screen "输入显示" 800x480
   Rectangle "矩形_2" at 16,42 size 105x25
      Appearance <- "工作台放松压检"
   Rectangle "矩形_1" at 16,14 size 105x25
      Appearance <- "工作台夹紧压检"
   Button "按钮_1" at 28,424 size 67x56; TextOn '滑块角度'; TextOff '滑块角度'
      on Click: ActivateScreen("滑块角度", 0)
   Button "按钮_2" at 96,424 size 67x56; TextOn '设备状态'; TextOff '设备状态'
      on Click: ActivateScreen("设备状态", 0)
   Button "按钮_3" at 163,424 size 71x55; TextOn '工作台操作'; TextOff '工作台操作'
      on Click: ActivateScreen("工作台操作", 0)
   Button "按钮_4" at 235,424 size 69x56; TextOn '气垫操作'; TextOff '气垫操作'
      on Click: ActivateScreen("气垫操作", 0)
   Button "按钮_5" at 304,423 size 66x57; TextOn '故障显示'; TextOff '故障显示'
      on Click: ActivateScreen("故障显示", 0)
   Button "按钮_6" at 371,423 size 73x57; TextOn '输出显示'; TextOff '输出显示'
      on Click: ActivateScreen("输出显示", 0)
   Button "按钮_7" at 445,422 size 66x58; TextOn '输入显示'; TextOff '输入显示'
      on Click: ActivateScreen("输入显示", 0)
   Button "按钮_8" at 514,423 size 68x56; TextOn '滑块调整'; TextOff '滑块调整'
      on Click: ActivateScreen("滑块调整", 0)
   Button "按钮_9" at 592,422 size 65x58; TextOn '报警信息'; TextOff '报警信息'
      on Click: ActivateScreen("报警信息", 0)
   TextField "文本域_1" at 18,20 size 103x17; Text '工作台夹紧压力'
   TextField "文本域_2" at 18,46 size 103x17; Text '工作台放松压力'
   Rectangle "矩形_3" at 16,98 size 105x25
      Appearance <- "平衡缸气压检测"
   Rectangle "矩形_4" at 16,70 size 105x25
      Appearance <- "故障复位"
   Rectangle "矩形_5" at 16,154 size 105x25
      Appearance <- "滑块调整选择"
   Rectangle "矩形_6" at 16,126 size 105x25
      Appearance <- "主电机启动接触器接通"
   Rectangle "矩形_7" at 16,210 size 105x25
      Appearance <- "气垫调整"
   Rectangle "矩形_8" at 16,182 size 105x25
      Appearance <- "行程"
   Rectangle "矩形_9" at 16,266 size 105x25
      Appearance <- "滑块向上"
   Rectangle "矩形_10" at 16,238 size 105x25
      Appearance <- "模具更换"
   TextField "文本域_11" at 36,76 size 61x17; Text '故障复位'
   TextField "文本域_3" at 19,104 size 103x17; Text '平衡缸气压检测'
   TextField "文本域_4" at 15,133 size 105x13; Text '主电机启动接触器接通'
   TextField "文本域_5" at 23,160 size 89x17; Text '滑块调整选择'
   TextField "文本域_6" at 48,188 size 33x17; Text '行程'
   TextField "文本域_7" at 33,215 size 61x17; Text '气垫调整'
   TextField "文本域_8" at 32,243 size 61x17; Text '模具更换'
   TextField "文本域_9" at 32,271 size 61x17; Text '滑块向上'
   Rectangle "矩形_11" at 16,294 size 105x25
      Appearance <- "滑块向下"
   Rectangle "矩形_12" at 16,322 size 105x25
      Appearance <- "停上死点"
   Rectangle "矩形_13" at 16,350 size 105x25
      Appearance <- "滑块调整过扭矩"
   TextField "文本域_10" at 32,300 size 61x17; Text '滑块向下'
   TextField "文本域_12" at 32,327 size 61x17; Text '停上死点'
   TextField "文本域_13" at 17,356 size 103x17; Text '滑块调整过扭矩'
   Rectangle "矩形_14" at 16,377 size 105x25
      Appearance <- "液压保护卸荷"
   TextField "文本域_14" at 23,383 size 89x17; Text '液压保护卸荷'
   Rectangle "矩形_15" at 132,42 size 105x25
      Appearance <- "爬梯开关"
   Rectangle "矩形_16" at 132,14 size 105x25
      Appearance <- "液压保护压力检测"
   Rectangle "矩形_17" at 132,98 size 105x25
      Appearance <- "润滑启动按钮"
   Rectangle "矩形_18" at 132,70 size 105x25
      Appearance <- "润滑停止按钮"
   Rectangle "矩形_19" at 132,154 size 105x25
      Appearance <- "平衡缸手动润滑按钮"
   Rectangle "矩形_20" at 132,126 size 105x25
      Appearance <- "气垫手动润滑按钮"
   Rectangle "矩形_21" at 132,210 size 105x25
      Appearance <- "液压保护复位2"
   Rectangle "矩形_22" at 132,182 size 105x25
      Appearance <- "液压保护复位1"
   Rectangle "矩形_23" at 132,266 size 105x25
      Appearance <- "模具松开按钮"
   Rectangle "矩形_24" at 132,238 size 105x25
      Appearance <- "模具夹紧按钮"
   Rectangle "矩形_25" at 132,294 size 105x25
      Appearance <- "模具更换转换"
   Rectangle "矩形_26" at 132,322 size 105x25
      Appearance <- "工作台夹紧"
   Rectangle "矩形_27" at 132,350 size 105x25
      Appearance <- "工作台松开"
   Rectangle "矩形_28" at 132,377 size 105x25
      Appearance <- "微调启动按钮"
   Rectangle "矩形_29" at 248,42 size 105x25
      Appearance <- "微调反转"
   Rectangle "矩形_30" at 248,14 size 105x25
      Appearance <- "微调正转"
   Rectangle "矩形_31" at 248,98 size 105x25
      Appearance <- "主电机启动1"
   Rectangle "矩形_32" at 248,70 size 105x25
      Appearance <- "主电机停止"
   Rectangle "矩形_33" at 248,154 size 105x25
      Appearance <- "主电机启动2"
   Rectangle "矩形_34" at 248,126 size 105x25
      Appearance <- "微调选择(1)"
   Rectangle "矩形_35" at 248,210 size 105x25
      Appearance <- "寸动闭点1"
   Rectangle "矩形_36" at 248,182 size 105x25
      Appearance <- "寸动开点1"
   Rectangle "矩形_37" at 248,266 size 105x25
      Appearance <- "寸动闭点2"
   Rectangle "矩形_38" at 248,238 size 105x25
      Appearance <- "寸动开点2"
   Rectangle "矩形_39" at 248,294 size 105x25
      Appearance <- "寸动选择"
   Rectangle "矩形_40" at 248,322 size 105x25
      Appearance <- "单次选择"
   Rectangle "矩形_41" at 248,350 size 105x25
      Appearance <- "连续选择"
   Rectangle "矩形_42" at 248,377 size 105x25
      Appearance <- "急停闭点"
   Rectangle "矩形_43" at 364,42 size 105x25
      Appearance <- "急停开点2"
   Rectangle "矩形_44" at 364,14 size 105x25
      Appearance <- "急停开点1"
   Rectangle "矩形_45" at 364,98 size 105x25
      Appearance <- "润滑油位低"
   Rectangle "矩形_46" at 364,70 size 105x25
      Appearance <- "润滑油位高"
   Rectangle "矩形_47" at 364,154 size 105x25
      Appearance <- "润滑低压2"
   Rectangle "矩形_48" at 364,126 size 105x25
      Appearance <- "润滑低压1"
   Rectangle "矩形_49" at 364,210 size 105x25
      Appearance <- "润滑高压"
   Rectangle "矩形_50" at 364,182 size 105x25
      Appearance <- "润滑低压3"
   Rectangle "矩形_51" at 364,266 size 105x25
      Appearance <- "滤油器堵塞2"
   Rectangle "矩形_52" at 364,238 size 105x25
      Appearance <- "滤油器堵塞1"
   Rectangle "矩形_53" at 364,294 size 105x25
      Appearance <- "滤油器堵塞3"
   Rectangle "矩形_54" at 364,322 size 105x25
      Appearance <- "工作台落到位前(1)"
   Rectangle "矩形_55" at 364,350 size 105x25
      Appearance <- "工作台落到位后(1)"
   Rectangle "矩形_56" at 364,377 size 105x25
      Appearance <- "气垫落到位"
   TextField "文本域_15" at 131,19 size 109x16; Text '液压保护压力检测'
   TextField "文本域_16" at 146,47 size 61x17; Text '爬梯开关'
   TextField "文本域_17" at 137,75 size 89x17; Text '润滑停止按钮'
   TextField "文本域_18" at 138,104 size 89x17; Text '润滑启动按钮'
   TextField "文本域_19" at 131,130 size 109x16; Text '气垫手动润滑按钮'
   TextField "文本域_20" at 128,159 size 113x15; Text '平衡缸手动润滑按钮'
   TextField "文本域_21" at 138,187 size 97x17; Text '液压保护复位1'
   TextField "文本域_22" at 137,215 size 97x17; Text '液压保护复位2'
   TextField "文本域_23" at 139,244 size 89x17; Text '模具夹紧按钮'
   TextField "文本域_24" at 139,272 size 89x17; Text '模具松开按钮'
   TextField "文本域_25" at 139,299 size 89x17; Text '模具更换转换'
   TextField "文本域_26" at 142,327 size 75x17; Text '工作台夹紧'
   TextField "文本域_27" at 141,354 size 75x17; Text '工作台松开'
   TextField "文本域_28" at 139,382 size 89x17; Text '微调启动按钮'
   TextField "文本域_29" at 267,20 size 61x17; Text '微调正转'
   TextField "文本域_30" at 267,47 size 61x17; Text '微调反转'
   TextField "文本域_31" at 261,75 size 75x17; Text '主电机停止'
   TextField "文本域_32" at 260,104 size 83x17; Text '主电机启动1'
   TextField "文本域_33" at 260,131 size 85x17; Text '微调选择(1)'
   TextField "文本域_34" at 262,159 size 83x17; Text '主电机启动2'
   TextField "文本域_35" at 267,188 size 69x17; Text '寸动开点1'
   TextField "文本域_36" at 267,216 size 69x17; Text '寸动闭点1'
   TextField "文本域_37" at 266,243 size 69x17; Text '寸动开点2'
   TextField "文本域_38" at 265,271 size 69x17; Text '寸动闭点2'
   TextField "文本域_39" at 268,299 size 61x17; Text '寸动选择'
   TextField "文本域_40" at 270,329 size 61x17; Text '单次选择'
   TextField "文本域_41" at 270,354 size 61x17; Text '连续选择'
   TextField "文本域_42" at 269,382 size 61x17; Text '急停闭点'
   TextField "文本域_43" at 382,20 size 69x17; Text '急停开点1'
   TextField "文本域_44" at 382,47 size 69x17; Text '急停开点2'
   TextField "文本域_45" at 379,75 size 75x17; Text '润滑油位高'
   TextField "文本域_46" at 379,104 size 75x17; Text '润滑油位低'
   TextField "文本域_47" at 381,132 size 69x17; Text '润滑低压1'
   TextField "文本域_48" at 381,158 size 69x17; Text '润滑低压2'
   TextField "文本域_49" at 381,187 size 69x17; Text '润滑低压3'
   TextField "文本域_50" at 384,215 size 61x17; Text '润滑高压'
   TextField "文本域_51" at 375,241 size 83x17; Text '滤油器堵塞1'
   TextField "文本域_52" at 374,272 size 83x17; Text '滤油器堵塞2'
   TextField "文本域_53" at 374,299 size 83x17; Text '滤油器堵塞3'
   TextField "文本域_54" at 361,328 size 103x17; Text '工作台落到位前'
   TextField "文本域_55" at 361,355 size 103x17; Text '工作台落到位后'
   TextField "文本域_56" at 375,382 size 75x17; Text '气垫落到位'

screen "输出显示" 800x480
   Button "按钮_1" at 28,424 size 67x56; TextOn '滑块角度'; TextOff '滑块角度'
      on Click: ActivateScreen("滑块角度", 0)
   Button "按钮_2" at 96,424 size 67x56; TextOn '设备状态'; TextOff '设备状态'
      on Click: ActivateScreen("设备状态", 0)
   Button "按钮_3" at 163,424 size 71x55; TextOn '工作台操作'; TextOff '工作台操作'
      on Click: ActivateScreen("工作台操作", 0)
   Button "按钮_4" at 235,424 size 69x56; TextOn '气垫操作'; TextOff '气垫操作'
      on Click: ActivateScreen("气垫操作", 0)
   Button "按钮_5" at 304,423 size 66x57; TextOn '故障显示'; TextOff '故障显示'
      on Click: ActivateScreen("故障显示", 0)
   Button "按钮_6" at 371,423 size 73x57; TextOn '输出显示'; TextOff '输出显示'
      on Click: ActivateScreen("输出显示", 0)
   Button "按钮_7" at 445,422 size 66x58; TextOn '输入显示'; TextOff '输入显示'
      on Click: ActivateScreen("输入显示", 0)
   Button "按钮_8" at 514,423 size 68x56; TextOn '滑块调整'; TextOff '滑块调整'
      on Click: ActivateScreen("滑块调整", 0)
   Button "按钮_9" at 592,422 size 65x58; TextOn '报警信息'; TextOff '报警信息'
      on Click: ActivateScreen("报警信息", 0)
   Rectangle "矩形_43" at 70,48 size 105x25
      Appearance <- "润滑油泵启动2"
   Rectangle "矩形_44" at 70,20 size 105x25
      Appearance <- "主电机正转DI1"
   Rectangle "矩形_45" at 70,104 size 105x25
      Appearance <- "KM3"
   Rectangle "矩形_46" at 70,76 size 105x25
      Appearance <- "M6 ?"
   Rectangle "矩形_47" at 70,160 size 105x25
      Appearance <- "气垫调整防粘连KM19"
   Rectangle "矩形_48" at 70,132 size 105x25
      Appearance <- "主电机启动JW1"
   Rectangle "矩形_49" at 70,216 size 105x25
      Appearance <- "气垫调整向下KM21"
   Rectangle "矩形_50" at 70,188 size 105x25
      Appearance <- "气垫调整向上KM20"
   Rectangle "矩形_51" at 70,272 size 105x25
      Appearance <- "滑块调整防粘连KM5"
   Rectangle "矩形_52" at 70,244 size 105x25
      Appearance <- "润滑油泵启动KM11"
   Rectangle "矩形_53" at 70,300 size 105x25
      Appearance <- "滑块向上KM6"
   Rectangle "矩形_54" at 70,328 size 105x25
      Appearance <- "滑块向下KM7"
   Rectangle "矩形_55" at 70,356 size 105x25
      Appearance <- "制动器阀"
   Rectangle "矩形_56" at 70,383 size 105x25
      Appearance <- "飞轮制动阀"
   TextField "文本域_1" at 71,26 size 99x17; Text '主电机正转DI1'
   TextField "文本域_2" at 72,54 size 97x17; Text '润滑油泵启动2'
   TextField "文本域_3" at 98,81 size 37x17; Text 'M6 ?'
   TextField "文本域_4" at 101,109 size 29x17; Text 'KM3'
   TextField "文本域_5" at 74,136 size 99x17; Text '主电机启动JW1'
   TextField "文本域_6" at 71,166 size 99x13; Text '气垫调整防粘连KM19'
   TextField "文本域_7" at 67,193 size 105x15; Text '气垫调整向上KM20'
   TextField "文本域_8" at 68,222 size 105x15; Text '气垫调整向下KM21'
   TextField "文本域_9" at 67,250 size 105x15; Text '润滑油泵启动KM11'
   TextField "文本域_10" at 67,277 size 110x15; Text '滑块调整防粘连KM5'
   TextField "文本域_11" at 78,306 size 85x17; Text '滑块向上KM6'
   TextField "文本域_12" at 78,333 size 85x17; Text '滑块向下KM7'
   TextField "文本域_13" at 87,361 size 61x17; Text '制动器阀'
   TextField "文本域_14" at 80,388 size 75x17; Text '飞轮制动阀'
   Rectangle "矩形_1" at 188,48 size 105x25
      Appearance <- "工作台放松阀(1)"
   Rectangle "矩形_2" at 188,20 size 105x25
      Appearance <- "工作台夹紧阀(1)"
   Rectangle "矩形_3" at 188,104 size 105x25
      Appearance <- "离合器阀"
   Rectangle "矩形_4" at 188,76 size 105x25
      Appearance <- "下死点指示(1)"
   Rectangle "矩形_5" at 188,160 size 105x25
      Appearance <- "KA41主电机正转"
   Rectangle "矩形_6" at 188,132 size 105x25
      Appearance <- "平衡缸润滑阀"
   Rectangle "矩形_7" at 188,216 size 105x25
      Appearance <- "润滑油位低指示"
   Rectangle "矩形_8" at 188,188 size 105x25
      Appearance <- "上死点指示"
   Rectangle "矩形_9" at 188,272 size 105x25
      Appearance <- "气垫润滑高压指示"
   Rectangle "矩形_10" at 188,244 size 105x25
      Appearance <- "润滑油位高指示"
   Rectangle "矩形_11" at 188,300 size 105x25
      Appearance <- "滤油器堵塞指示"
   Rectangle "矩形_12" at 188,328 size 105x25
      Appearance <- "滑块向下KM7"
   Rectangle "矩形_13" at 188,356 size 105x25
      Appearance <- "制动器阀"
   Rectangle "矩形_14" at 188,383 size 105x25
      Appearance <- "飞轮制动阀"
   TextField "文本域_15" at 184,26 size 113x17; Text '工作台夹紧阀(1)'
   TextField "文本域_16" at 183,51 size 113x17; Text '工作台放松阀(1)'
   TextField "文本域_17" at 190,80 size 99x17; Text '下死点指示(1)'
   TextField "文本域_18" at 203,109 size 61x17; Text '离合器阀'
   TextField "文本域_19" at 194,137 size 89x17; Text '平衡缸润滑阀'
   TextField "文本域_20" at 187,164 size 107x17; Text 'KA41主电机正转'
   TextField "文本域_21" at 200,193 size 75x17; Text '上死点指示'
   TextField "文本域_22" at 185,221 size 103x17; Text '润滑油位低指示'
   TextField "文本域_23" at 187,250 size 103x17; Text '润滑油位高指示'
   TextField "文本域_24" at 181,279 size 117x17; Text '气垫润滑高压指示'
   TextField "文本域_25" at 188,306 size 103x17; Text '滤油器堵塞指示'

screen "故障显示" 800x480
   Button "按钮_1" at 28,424 size 67x56; TextOn '滑块角度'; TextOff '滑块角度'
      on Click: ActivateScreen("滑块角度", 0)
   Button "按钮_2" at 96,424 size 67x56; TextOn '设备状态'; TextOff '设备状态'
      on Click: ActivateScreen("设备状态", 0)
   Button "按钮_3" at 163,424 size 71x55; TextOn '工作台操作'; TextOff '工作台操作'
      on Click: ActivateScreen("工作台操作", 0)
   Button "按钮_4" at 235,424 size 69x56; TextOn '气垫操作'; TextOff '气垫操作'
      on Click: ActivateScreen("气垫操作", 0)
   Button "按钮_5" at 304,423 size 66x57; TextOn '故障显示'; TextOff '故障显示'
      on Click: ActivateScreen("故障显示", 0)
   Button "按钮_6" at 371,423 size 73x57; TextOn '输出显示'; TextOff '输出显示'
      on Click: ActivateScreen("输出显示", 0)
   Button "按钮_7" at 445,422 size 66x58; TextOn '输入显示'; TextOff '输入显示'
      on Click: ActivateScreen("输入显示", 0)
   Button "按钮_8" at 514,423 size 68x56; TextOn '滑块调整'; TextOff '滑块调整'
      on Click: ActivateScreen("滑块调整", 0)
   Button "按钮_9" at 592,422 size 65x58; TextOn '报警信息'; TextOff '报警信息'
      on Click: ActivateScreen("报警信息", 0)

screen "工作台操作" 800x480
   Button "按钮_1" at 28,424 size 67x56; TextOn '滑块角度'; TextOff '滑块角度'
      on Click: ActivateScreen("滑块角度", 0)
   Button "按钮_2" at 96,424 size 67x56; TextOn '设备状态'; TextOff '设备状态'
      on Click: ActivateScreen("设备状态", 0)
   Button "按钮_3" at 163,424 size 71x55; TextOn '工作台操作'; TextOff '工作台操作'
      on Click: ActivateScreen("工作台操作", 0)
   Button "按钮_4" at 235,424 size 69x56; TextOn '气垫操作'; TextOff '气垫操作'
      on Click: ActivateScreen("气垫操作", 0)
   Button "按钮_5" at 304,423 size 66x57; TextOn '故障显示'; TextOff '故障显示'
      on Click: ActivateScreen("故障显示", 0)
   Button "按钮_6" at 371,423 size 73x57; TextOn '输出显示'; TextOff '输出显示'
      on Click: ActivateScreen("输出显示", 0)
   Button "按钮_7" at 445,422 size 66x58; TextOn '输入显示'; TextOff '输入显示'
      on Click: ActivateScreen("输入显示", 0)
   TextField "文本域_1" at 47,79 size 125x27; Text '工作台松开'
   TextField "文本域_2" at 53,142 size 125x27; Text '工作台夹紧'
   Circle "圆_5" at 530,81 size 27x27
      Appearance <- "工作台放松阀(1)"
   TextField "文本域_10" at 502,111 size 83x16; Text '工作台松开阀'
   Circle "圆_7" at 428,81 size 27x27
      Appearance <- "工作台松开"
   TextField "文本域_12" at 405,111 size 70x16; Text '工作台松开'
   Circle "圆_8" at 222,81 size 27x27
      Appearance <- "上死点指示"
   TextField "文本域_13" at 215,111 size 44x16; Text '上死点'
   Circle "圆_9" at 630,81 size 27x27
      Appearance <- "工作台放松压检"
   TextField "文本域_14" at 597,111 size 96x16; Text '工作台松开压力'
   Circle "圆_6" at 718,81 size 27x27
      Appearance <- "工作台放松OK"
   TextField "文本域_11" at 693,111 size 84x16; Text '工作台松开OK'
   Circle "圆_14" at 325,141 size 27x27
      Appearance <- "工作台夹紧"
   TextField "文本域_19" at 304,171 size 70x16; Text '工作台夹紧'
   Circle "圆_15" at 222,141 size 27x27
      Appearance <- "工作台落到位"
   TextField "文本域_20" at 197,171 size 83x16; Text '工作台落到位'
   Circle "圆_16" at 428,141 size 27x27
      Appearance <- "工作台夹紧阀(1)"
   TextField "文本域_21" at 402,171 size 83x16; Text '工作台夹紧阀'
   Circle "圆_1" at 530,141 size 27x27
      Appearance <- "工作台夹紧压检"
   TextField "文本域_3" at 497,171 size 96x16; Text '工作台夹紧压力'
   Circle "圆_2" at 619,141 size 27x27
      Appearance <- "工作台-夹紧OK"
   TextField "文本域_4" at 594,171 size 84x16; Text '工作台夹紧OK'
   Button "按钮_8" at 514,423 size 68x56; TextOn '滑块调整'; TextOff '滑块调整'
      on Click: ActivateScreen("滑块调整", 0)
   Button "按钮_9" at 592,422 size 65x58; TextOn '报警信息'; TextOff '报警信息'
      on Click: ActivateScreen("报警信息", 0)
   Circle "圆_3" at 325,82 size 27x27
      Appearance <- "气垫落到位"
   TextField "文本域_5" at 304,112 size 70x16; Text '气垫落到位'

screen "气垫操作" 800x480
   Button "按钮_1" at 28,424 size 67x56; TextOn '滑块角度'; TextOff '滑块角度'
      on Click: ActivateScreen("滑块角度", 0)
   Button "按钮_2" at 96,424 size 67x56; TextOn '设备状态'; TextOff '设备状态'
      on Click: ActivateScreen("设备状态", 0)
   Button "按钮_3" at 163,424 size 71x55; TextOn '工作台操作'; TextOff '工作台操作'
      on Click: ActivateScreen("工作台操作", 0)
   Button "按钮_4" at 235,424 size 69x56; TextOn '气垫操作'; TextOff '气垫操作'
      on Click: ActivateScreen("气垫操作", 0)
   Button "按钮_5" at 304,423 size 66x57; TextOn '故障显示'; TextOff '故障显示'
      on Click: ActivateScreen("故障显示", 0)
   Button "按钮_6" at 371,423 size 73x57; TextOn '输出显示'; TextOff '输出显示'
      on Click: ActivateScreen("输出显示", 0)
   Button "按钮_7" at 445,422 size 66x58; TextOn '输入显示'; TextOff '输入显示'
      on Click: ActivateScreen("输入显示", 0)
   Button "按钮_8" at 514,423 size 68x56; TextOn '滑块调整'; TextOff '滑块调整'
      on Click: ActivateScreen("滑块调整", 0)
   Button "按钮_9" at 592,422 size 65x58; TextOn '报警信息'; TextOff '报警信息'
      on Click: ActivateScreen("报警信息", 0)
   TextField "文本域_1" at 55,82 size 101x27; Text '气垫上调'
   TextField "文本域_2" at 58,142 size 101x27; Text '气垫下调'
   Circle "圆_8" at 295,81 size 27x27
      Appearance <- "上死点指示"
   TextField "文本域_13" at 288,111 size 44x16; Text '上死点'
   Circle "圆_3" at 358,82 size 27x27
      Appearance <- "气垫落到位"
   TextField "文本域_5" at 337,112 size 70x16; Text '气垫落到位'
   Circle "圆_1" at 296,146 size 27x27
      Appearance <- "上死点指示"
   TextField "文本域_3" at 289,176 size 44x16; Text '上死点'
   Circle "圆_2" at 359,147 size 27x27
      Appearance <- "气垫落到位"
   TextField "文本域_4" at 338,177 size 70x16; Text '气垫落到位'
   Circle "圆_4" at 427,82 size 27x27
      Appearance <- "气垫调整"
   TextField "文本域_6" at 410,112 size 57x16; Text '气垫调整'
   Circle "圆_6" at 496,82 size 27x27
      Appearance <- "气垫调整向上KM20"
   TextField "文本域_8" at 481,112 size 57x16; Text '气垫向上'
   Circle "圆_7" at 497,147 size 27x27
      Appearance <- "气垫调整向下KM21"
   TextField "文本域_9" at 483,177 size 57x16; Text '气垫向下'
   Button "按钮_10" at 8,8 size 96x32; TextOff 'Text'
   Button "按钮_11" at 187,240 size 102x89; TextOff '气垫向上'
      Appearance <- "气垫向上调整"
      on Press: function_b14e0dd5("气垫向上调整", 0)
   Button "按钮_12" at 323,240 size 102x89; TextOff '气垫向下'
      Appearance <- "气垫向下调整"
      on Press: function_b14e0dd5("气垫向下调整", 0)
   Circle "圆_5" at 430,147 size 27x27
      Appearance <- "气垫调整"
   TextField "文本域_7" at 413,177 size 57x16; Text '气垫调整'
   Circle "圆_15" at 232,147 size 27x27
      Appearance <- "工作台落到位"
   TextField "文本域_20" at 207,177 size 83x16; Text '工作台落到位'
   Circle "圆_9" at 230,81 size 27x27
      Appearance <- "工作台落到位"
   TextField "文本域_10" at 205,111 size 83x16; Text '工作台落到位'

screen "滑块调整" 800x480
   Button "按钮_1" at 28,424 size 67x56; TextOn '滑块角度'; TextOff '滑块角度'
      on Click: ActivateScreen("滑块角度", 0)
   Button "按钮_2" at 96,424 size 67x56; TextOn '设备状态'; TextOff '设备状态'
      on Click: ActivateScreen("设备状态", 0)
   Button "按钮_3" at 163,424 size 71x55; TextOn '工作台操作'; TextOff '工作台操作'
      on Click: ActivateScreen("工作台操作", 0)
   Button "按钮_4" at 235,424 size 69x56; TextOn '气垫操作'; TextOff '气垫操作'
      on Click: ActivateScreen("气垫操作", 0)
   Button "按钮_5" at 304,423 size 66x57; TextOn '故障显示'; TextOff '故障显示'
      on Click: ActivateScreen("故障显示", 0)
   Button "按钮_6" at 371,423 size 73x57; TextOn '输出显示'; TextOff '输出显示'
      on Click: ActivateScreen("输出显示", 0)
   Button "按钮_7" at 445,422 size 66x58; TextOn '输入显示'; TextOff '输入显示'
      on Click: ActivateScreen("输入显示", 0)
   Button "按钮_8" at 514,423 size 68x56; TextOff '滑块调整'
      on Click: ActivateScreen("滑块调整", 0)
   TextField "文本域_1" at 157,34 size 61x29; Text '1100'
   TextField "文本域_2" at 26,34 size 109x29; Text '滑块上限'
   TextField "文本域_3" at 158,107 size 47x29; Text '670'
   TextField "文本域_4" at 27,107 size 109x29; Text '滑块下限'
   TextField "文本域_6" at 268,33 size 135x29; Text '滑块当前值'
   TextField "文本域_8" at 270,108 size 135x29; Text '滑块设定值'
   TextField "文本域_9" at 580,184 size 149x27; Text '滑块高度设置'
   IOField "I/O 域_4" at 603,234 size 103x47; FormatPattern 9999
      ProcessValue <- "横梁编码器 _DB_+0.8"
   Circle "圆_1" at 584,30 size 39x39
      Appearance <- "滑块调整手动/自动"
   Circle "圆_2" at 690,31 size 39x39
      Appearance <- "滑块调整手动/自动"
   TextField "文本域_16" at 583,76 size 41x21; Text '手动'
   TextField "文本域_19" at 689,76 size 41x21; Text '自动'
   IOField "I/O 域_1" at 414,102 size 103x47; FormatPattern 9999
      ProcessValue <- "横梁编码器 _DB_+0.8"
   IOField "I/O 域_2" at 414,33 size 103x47; FormatPattern 9999
      ProcessValue <- "ECamdata _DB_D107"
   Switch "开关_1" at 600,93 size 120x56; CaptionText 'Switch'; TextOff '手动'; TextOn '自动'
      on SwitchOff: ResetBit("滑块调整手动/自动")
      on SwitchOn: SetBit("滑块调整手动/自动")
      Appearance <- "滑块调整自动选择"
   TextField "文本域_5" at 599,150 size 123x21; Text '手动/自动调整'
   Button "按钮_9" at 612,315 size 96x58; TextOff '自动调整开始'
      on Press: SetBit("滑块调整自动选择")
      Appearance <- "滑块调整自动选择"
      on Release: ResetBit("滑块调整自动选择")
   Button "按钮_10" at 592,422 size 65x58; TextOn '报警信息'; TextOff '报警信息'
      on Click: ActivateScreen("报警信息", 0)
   TextField "文本域_7" at 157,177 size 47x29; Text '800'
   TextField "文本域_10" at 26,177 size 109x29; Text '滑块行程'

screen "报警信息" 800x480
   AlarmView "报警视图_1" at 10,90 size 780x331
   Clock "时钟_1" at 630,64 size 164x20
   GraphicView "图形视图_2" at 2,9 size 78x46; Picture "方鼎LOGO"
   TextField "文本域_5" at 222,19 size 365x33; Text '湖北方鼎科技发展有限公司'
   TextField "文本域_3" at 710,9 size 75x21; Text 'SIEMENS'
   TextField "文本域_4" at 702,37 size 93x17; Text 'SIMATIC HMI'
   TextField "文本域_1" at 325,62 size 109x29; Text '报警信息'
   Button "按钮_1" at 28,424 size 67x56; TextOn '滑块角度'; TextOff '滑块角度'
      on Click: ActivateScreen("滑块角度", 0)
   Button "按钮_2" at 96,424 size 67x56; TextOn '设备状态'; TextOff '设备状态'
      on Click: ActivateScreen("设备状态", 0)
   Button "按钮_3" at 163,424 size 71x55; TextOn '工作台操作'; TextOff '工作台操作'
      on Click: ActivateScreen("工作台操作", 0)
   Button "按钮_4" at 235,424 size 69x56; TextOn '气垫操作'; TextOff '气垫操作'
      on Click: ActivateScreen("气垫操作", 0)
   Button "按钮_5" at 304,423 size 66x57; TextOn '故障显示'; TextOff '故障显示'
      on Click: ActivateScreen("故障显示", 0)
   Button "按钮_6" at 371,423 size 73x57; TextOn '输出显示'; TextOff '输出显示'
      on Click: ActivateScreen("输出显示", 0)
   Button "按钮_7" at 445,422 size 66x58; TextOn '输入显示'; TextOff '输入显示'
      on Click: ActivateScreen("输入显示", 0)
   Button "按钮_8" at 514,423 size 68x56; TextOn '滑块调整'; TextOff '滑块调整'
      on Click: ActivateScreen("滑块调整", 0)
   Button "按钮_9" at 592,422 size 65x58; TextOn '报警信息'; TextOff '报警信息'
      on Click: ActivateScreen("报警信息", 0)
*)